ABB RobotStudio station: Lab1.13_20210910-122509.rsstn

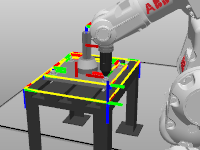
Station Lab1.12 (saved by RobotStudio 21.2.9526.0)
Controller IRB140_6_81
  mechanical unit ROB_1: IRB140_6_81_C_03, 6 joints, base frame (0, 0, 0) mm
Layout (positions relative to the parent item):
  - IRB140_6_81_C_03 [mechanism, from Robots\IRB140_6_81_C_G_03.rslib] at (0, 0, 0) mm; joint values [0.1974, -0.0317, 0.5823, 0, 1.0202, -2.9442] (rad or m)
  - table_and_fixture_140 [part, from Training Objects\propeller_table.rslib] at (300, 225, 0) mm, rotated rx 0 ry 0 rz -90 deg
  - UISpenholder [mechanism, from RS1\UISpenholder.rslib] at (375, 75, 448) mm, rotated rx -180 ry 0 rz 0 deg
Attachment: WobjTable is attached to table_and_fixture_140
Attachment: UISpenholder is attached to IRB140_6_81_C_03 / Link6
Collision set CollisionSet_1: UISpenholder against table_and_fixture_140, near miss 0 m
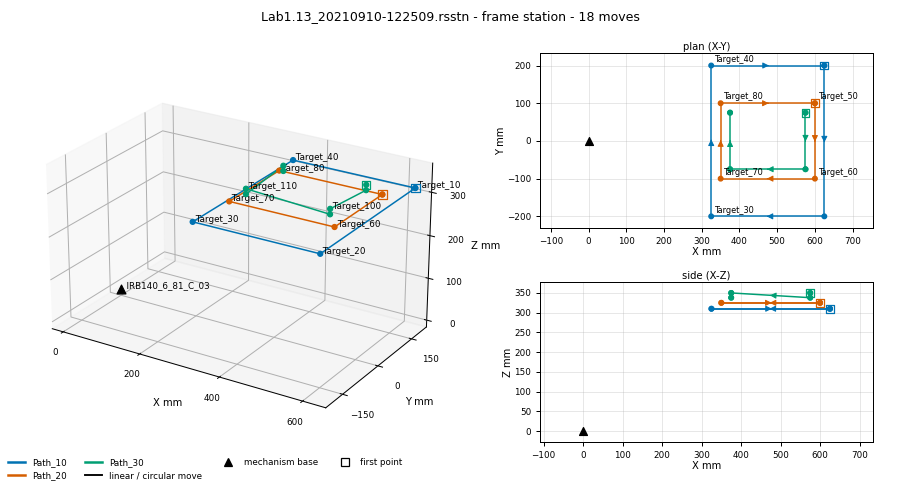
[picture p0: tool path of Lab1.13_20210910-122509.rsstn in frame station, 18 of 18 moves have a stored position in this frame; points joined in program order, loops and branches not executed]
Targets, tools, work objects and paths stored in the station, written as RAPID:
! task T_ROB1
MODULE Module1
  TASK PERS wobjdata WobjTable:=[FALSE,TRUE,"",[[475,625,2],[0.707106781,0,0,-0.707106781]],[[425,-150,308],[1,0,0,0]]];
  CONST robtarget Target_10:=[[0,300,0],[0,1,0,0],[0,0,0,0],[9E+09,9E+09,9E+09,9E+09,9E+09,9E+09]];
  CONST robtarget Target_20:=[[400,300,0],[0,-0.707106781,0.707106781,0],[-1,0,-1,0],[9E+09,9E+09,9E+09,9E+09,9E+09,9E+09]];
  CONST robtarget Target_30:=[[400,0,0],[0,0,1,0],[-1,0,0,0],[9E+09,9E+09,9E+09,9E+09,9E+09,9E+09]];
  CONST robtarget Target_40:=[[0,0,0],[0,1,0,0],[0,0,-2,0],[9E+09,9E+09,9E+09,9E+09,9E+09,9E+09]];
  CONST robtarget Target_50:=[[100,275,15],[0,1,0,0],[0,0,0,0],[9E+09,9E+09,9E+09,9E+09,9E+09,9E+09]];
  CONST robtarget Target_60:=[[300,275,15],[0,-0.707106781,0.707106781,0],[-1,0,-1,0],[9E+09,9E+09,9E+09,9E+09,9E+09,9E+09]];
  CONST robtarget Target_70:=[[300,25,15],[0,0,1,0],[-1,0,0,0],[9E+09,9E+09,9E+09,9E+09,9E+09,9E+09]];
  CONST robtarget Target_80:=[[100,25,15],[0,1,0,0],[0,0,-2,0],[9E+09,9E+09,9E+09,9E+09,9E+09,9E+09]];
  CONST robtarget Target_90:=[[125,250,40],[0,1,0,0],[0,0,0,0],[9E+09,9E+09,9E+09,9E+09,9E+09,9E+09]];
  CONST robtarget Target_100:=[[275,250,40],[0,-0.707106781,0.707106781,0],[-1,0,-1,0],[9E+09,9E+09,9E+09,9E+09,9E+09,9E+09]];
  CONST robtarget Target_110:=[[275,50,40],[0,0,1,0],[-1,0,0,0],[9E+09,9E+09,9E+09,9E+09,9E+09,9E+09]];
  CONST robtarget Target_120:=[[125,50,40],[0,0.707106781,0.707106781,0],[0,0,-2,0],[9E+09,9E+09,9E+09,9E+09,9E+09,9E+09]];
  CONST robtarget Target_90_2:=[[125,250,28],[0,1,0,0],[0,0,-1,0],[9E+09,9E+09,9E+09,9E+09,9E+09,9E+09]];
  CONST robtarget Target_100_2:=[[275,250,28],[0,-0.707106781,0.707106781,0],[-1,0,-1,0],[9E+09,9E+09,9E+09,9E+09,9E+09,9E+09]];
  CONST robtarget Target_110_2:=[[275,50,28],[0,0,1,0],[-1,0,0,0],[9E+09,9E+09,9E+09,9E+09,9E+09,9E+09]];
  CONST robtarget Target_120_2:=[[125,50,28],[0,0.707106781,0.707106781,0],[0,0,-2,0],[9E+09,9E+09,9E+09,9E+09,9E+09,9E+09]];
  CONST robtarget Target_Center:=[[200,150,183],[0,1,0,0],[0,0,0,0],[9E+09,9E+09,9E+09,9E+09,9E+09,9E+09]];
  PROC Path_10()
    MoveL Target_10,v1000,z5,UISpenholder\WObj:=WobjTable;
    MoveL Target_20,v1000,z5,UISpenholder\WObj:=WobjTable;
    MoveL Target_30,v1000,z5,UISpenholder\WObj:=WobjTable;
    MoveL Target_40,v1000,z5,UISpenholder\WObj:=WobjTable;
    MoveL Target_10,v1000,z5,UISpenholder\WObj:=WobjTable;
  ENDPROC
  PROC Path_20()
    MoveL Target_50,v1000,z5,UISpenholder\WObj:=WobjTable;
    MoveL Target_60,v1000,z5,UISpenholder\WObj:=WobjTable;
    MoveL Target_70,v1000,z5,UISpenholder\WObj:=WobjTable;
    MoveL Target_80,v1000,z5,UISpenholder\WObj:=WobjTable;
    MoveL Target_50,v1000,z5,UISpenholder\WObj:=WobjTable;
  ENDPROC
  PROC Path_30()
    MoveL Target_90,v1000,z100,UISpenholder\WObj:=WobjTable;
    MoveL Target_90_2,v1000,z100,UISpenholder\WObj:=WobjTable;
    MoveL Target_100,v1000,z100,UISpenholder\WObj:=WobjTable;
    MoveL Target_100_2,v1000,z100,UISpenholder\WObj:=WobjTable;
    MoveL Target_110,v1000,z100,UISpenholder\WObj:=WobjTable;
    MoveL Target_110_2,v1000,z100,UISpenholder\WObj:=WobjTable;
    MoveL Target_120,v1000,z100,UISpenholder\WObj:=WobjTable;
    MoveL Target_120_2,v1000,z100,UISpenholder\WObj:=WobjTable;
  ENDPROC
ENDMODULE

! task T_ROB1
MODULE CalibData
  PERS tooldata Pen_TCP:=[TRUE,[[110,0,140],[0.707106781,0,0.707106781,0]],[1,[10.7435139,0,140],[1,0,0,0],0,0,0]];
  PERS tooldata UISpenholder:=[TRUE,[[0,0,110],[1,0,0,0]],[1,[0,0,1],[1,0,0,0],0,0,0]];
ENDMODULE

